(*
SPDX-FileCopyrightText: Â© 2026 Oleksandr Tiutyk <trofimich@gmail.com>
SPDX-License-Identifier: MIT
License: https://opensource.org/license/mit
*)

(*!
<summary>Represents a child automation component with an overridable simulation mode.</summary>
*)

INTERFACE IChildSimulatable EXTENDS ISimulatable

(*!
<summary>Gets the simulation mode override setting for this child component.</summary>
*)
{attribute 'monitoring' := 'call'}
PROPERTY SimulationModeOverride : SIMULATION_MODE_OVERRIDE
GET
END_GET
END_PROPERTY

END_INTERFACE

(* stored: Version 1.1.0.1
   Itf IChildSimulatable: Id {b3d832ce-36cd-4ef3-8946-ef433813ca83}
   Property SimulationModeOverride: Id {3d124263-0bc7-4bdf-92ab-74226bdb0bea}
   Get Get: Id {69346a08-4864-4225-81f4-0c0162415556} *)
